// TIA Portal V19 export
ORGANIZATION_BLOCK "Main"   // OB1, STL, ProgramCycle
TITLE = Zyklus
{ S7_Optimized_Access := 'FALSE' }
AUTHOR : MS
// stored: AutoNumber false
   VAR_TEMP
      OB1_EV_CLASS : Byte;   // Bits 0-3 = 1 (Coming event), Bits 4-7 = 1 (Event class 1)
      OB1_SCAN_1 : Byte;   // 1 (Cold restart scan 1 of OB 1), 3 (Scan 2-n of OB 1)
      OB1_PRIORITY : Byte;   // 1 (Priority of 1 is lowest)
      OB1_OB_NUMBR : Byte;   // 1 (Organization block 1, OB1)
      OB1_RESERVED_1 : Byte;   // Reserved for system
      OB1_RESERVED_2 : Byte;   // Reserved for system
      OB1_PREV_CYCLE : Int;   // Cycle time of previous OB1 scan (milliseconds)
      OB1_MIN_CYCLE : Int;   // Minimum cycle time of OB1 (milliseconds)
      OB1_MAX_CYCLE : Int;   // Maximum cycle time of OB1 (milliseconds)
      OB1_DATE_TIME : Date_And_Time;   // Date and time OB1 started
   END_VAR
BEGIN

NETWORK
TITLE = 
//-------------------------
//Zykluszeit merken
//-------------------------
      L     #OB1_PREV_CYCLE;
      T     "DI_FW_MANAGER".akt_CT;
      L     "DI_FW_MANAGER".max_CT;
      <I;
      JC    writ;
      L     "DI_FW_MANAGER".akt_CT;
writ: T     "DI_FW_MANAGER".max_CT;
//-------------------------
//neue Anlagenkonfiguration
//-------------------------
      AN    "DB_ANLAGE".BA.newConfig;
      JC    nCfg;
      CALL  "FC_newConfig"
      ( Anlauf := FALSE
      );
nCfg: NOP   0;

//------------------------------
//Flankenauswertung Taktmerker
//------------------------------
      CALL  "Taktmerker";
//-------------------------
//Wochenschaltuhr
//-------------------------
      CALL  "Schaltuhr";
      CALL  "Uhrzeit_WSU", "Uhrzeit";

//------------------------------
//Zeiten aktualisieren
//------------------------------
      A     "Imp_1Hz";
      CC    "FC_EXPO_TIME";
//-------------------------
//PNOZ-Kommunikation
//-------------------------
      CALL  "Komm_PNOZ";
//-------------------------
//Eingänge/Eingaben lesen
//-------------------------
      CALL  "FC_DP_Error";
      CALL  "FU_Read";
      CALL  "FC_INPUT";
      CALL  "FC_SIMULATION";
//-------------------------
//Analogwerterfassung
//-------------------------
      CALL  "Analogeingabe";
//-------------------------
//Betriebsarten setzen
//-------------------------
      CALL  "BA_WXL";
//-------------------------
//Optimierung
//-------------------------
      CALL  "FC_Optimierung";
//-------------------------
//WT-Verwaltung
//-------------------------
      CALL  "FC_WT_MANAGER";
//-------------------------
//Fahrwagenverwaltung
//-------------------------
      CALL  "FC_Hilfsfuntionen";
//----------------------------------
//Pos-Reservierung überarbeiten
//----------------------------------
      CALL  "FC_FW_RES_QZ";
//----------------------------------
// FW-Verwaltung (nur bei Auftrag)
//----------------------------------
      CALL  "FB_FW_Auftrag", "DI_FW_Auftrag_DB";
//-------------------------
//Fahrwagen bearbeiten
//-------------------------
      CALL  "FB_FW_MANAGER", "DI_FW_MANAGER"
      ( CallDBNr := 
      );
//-------------------------
//Badverwaltung
//-------------------------
      CALL  "FC_Pos_Manager";
//-------------------------
//Ladungszähler
//-------------------------
      CALL  "FC_Zaehler";
      CALL  "FC_DoPu";
//-------------------------
//Anlagenfunktionen
//-------------------------
      CALL  "Peripherie";
      CALL  "FC_Niveau_St";
//-------------------------
//Alarmbehandlung gesamt
//-------------------------
      CALL  "Alarme";

//-------------------------
//Ausgänge schreiben
//-------------------------
      CALL  "FC_OUTPUT";
      CALL  "FU_Write";
//-------------------------
//Daten bereitstellen
//-------------------------
      CALL  "FC_Copy_Daten_Heraeus";

      BE;
END_ORGANIZATION_BLOCK
